FUNCTION_BLOCK EM_OutfeedModule EXTENDS CommonModule IMPLEMENTS I_OutfeedModule
VAR
	//Components
	Axis : FB_Component_BasicAxis;

	//
	_CmdOutfeed : ST_OutfeedCommand;
	_StsOutfeed : ST_OutfeedStatus;
	_CfgOutfeed : ST_OutfeedConfig;
	_RcpOutfeed : ST_OutfeedRecipe;

	//Test Vars
	Homed : BOOL;
END_VAR

PROPERTY CfgOutfeed : REFERENCE TO ST_OutfeedConfig
GET
CfgOutfeed REF= _CfgOutfeed;
END_GET
END_PROPERTY

PROPERTY CmdOutfeed : REFERENCE TO ST_OutfeedCommand
GET
CmdOutfeed REF= _CmdOutfeed;
END_GET
END_PROPERTY

METHOD PUBLIC CyclicLogic
IF NOT _InitComplete THEN
	_InitComplete := Initialize();
	RETURN;
END_IF

SUPER^.CyclicLogic();
END_METHOD

//! @summary This method contains code which will execute when this PackML module is in the <b>Execute</b> state
METHOD PROTECTED Execute
(*! <description> <b>The base implementation of this method is empty. User must override this method to provide functionality.</b>
<table> 
	<tr>
		<th> Previous State </th>
		<th> Transition In </th>
		<th> Transition Out </th>
		<th> Next State  </th> 
	</tr>
	<tr>
		<td> Starting<b>-or-</b>Unholding <b>-or-</b>Unsuspending</td>
		<td> State Complete<i>(Starting<b>-or-</b>Unholding<b>-or-</b>Unsuspending)</i></td> 
		<td> State Complete<b>-or-</b>Hold Command<b>-or-</b>Suspend Command</td>
		<td> Completing<b>-or-</b>Holding<b>-or-</b>Suspending</td>
	</tr>
</table>
This method is called as required by <c>StateControl()</c>
</description> 

*)
VAR
END_VAR
CASE _CurrentMode OF
	E_PMLCustomMode.Production:
		CASE DescendantSequenceState OF
			0:
				IF _StsOutfeed.ProductAtReady THEN
					DescendantSequenceState := DescendantSequenceState + 10;
				END_IF

			10:
				IF Axis.MoveVelocity(10.0, 0) THEN
					DescendantSequenceState := DescendantSequenceState + 10;
				END_IF

			20:
				IF Axis.Axis.Status.Moving THEN
					_StsOutfeed.ProductAtReady	:= FALSE;
					_StsOutfeed.ConveyorRunning := TRUE;
				END_IF

				IF _StsOutfeed.ProductRemoved THEN
					_CmdOutfeed.StopConveyor := FALSE;
					Axis.Stop();
					DescendantSequenceState := DescendantSequenceState + 10;
				END_IF

			30:
				IF Axis.Axis.Status.NotMoving THEN
					_StsOutfeed.ConveyorRunning := FALSE;
					DescendantSequenceState		:= 0;
				END_IF
		END_CASE

	E_PMLCustomMode.Home:
		CASE DescendantSequenceState OF
			0:
				IF _CmdCommon.Home AND NOT _StsCommon.Homed THEN
					_CmdCommon.Home := FALSE;
					Axis.Home();
					DescendantSequenceState := DescendantSequenceState + 10;
				END_IF

			10:
				IF Axis.Axis.Status.Homed THEN
					_StsCommon.Homed := TRUE;
				END_IF
		END_CASE
END_CASE

SUPER^.Execute();
END_METHOD

METHOD PROTECTED Initialize : BOOL
VAR
	i: UDINT;
END_VAR
Initialize := FALSE;
CASE DescendantSequenceState OF
	0: //Register Modules

		//Register Components
		RegisterComponent(Axis);

		//I_CommonModuleBase

		//I_CommonComponent
		ipComponents[1] := Axis;

		//Setup Config
		_LogModeChanges			:= FALSE;
		_LogStateChanges		:= FALSE;
		DescendantSequenceState := DescendantSequenceState + 10;

	10:
		// Copy Mode names
		FOR i := 1 TO 10 DO
			ModeNames[i] := F_UnitModeToString(UDINT_TO_DINT(i));
		END_FOR

		DescendantSequenceState := DescendantSequenceState + 10;

	20:
		//Initialize_Recipes();
		DescendantSequenceState := DescendantSequenceState + 10;

	30: // Call the Super 
		IF SUPER^.Initialize() THEN
			DescendantSequenceState := DescendantSequenceState + 10;
		END_IF

	40:
		Initialize := TRUE;
END_CASE
END_METHOD

PROPERTY RcpOutfeed : REFERENCE TO ST_OutfeedRecipe
GET
RcpOutfeed REF= _RcpOutfeed;
END_GET
END_PROPERTY

PROPERTY StsOutfeed : REFERENCE TO ST_OutfeedStatus
GET
StsOutfeed REF= _StsOutfeed;
END_GET
END_PROPERTY

END_FUNCTION_BLOCK

(* stored: Version 1.1.0.1, ProductVersion 3.1.4024.12
   POU EM_OutfeedModule: Id {7cfe66d8-35ba-4314-bc5b-79de6dfce221}, SpecialFunc None
   Folder I_CyclicLogic: Id {bff73ff0-91fb-43bc-8249-92d4b9647678}
   Folder I_OutfeedModule: Id {69613287-f892-473e-b1d8-0484c46e7d3a}
   Folder Initialize: Id {2f6fe5d0-4ad8-4db5-bcbb-919a2371bcc0}
   Folder Waiting: Id {90aacb5d-d031-4a9a-a8b9-804c40c70e47}
   Property CfgOutfeed: Id {a44dd973-0916-4949-a737-65d3485b91ec}
   Get Get: Id {319902ff-1362-472b-b229-c462e2493a5e}
   Property CmdOutfeed: Id {4c76f708-fd44-49ee-89dc-ce3046ef3f80}
   Get Get: Id {b3b04fb8-826d-4de2-b263-f0bc53875584}
   Method CyclicLogic: Id {4340cd9c-c928-4e0a-bb64-e13a6fc3c8ca}
   Method Execute: Id {72fd1940-d387-4987-ac34-491b6521b66b}
   Method Initialize: Id {5233c20d-7b9b-4059-b797-40c895a2027a}
   Property RcpOutfeed: Id {0b12ebb9-62cb-4cc2-b1ed-ede402f73212}
   Get Get: Id {b53521d8-ac70-4d27-bdae-fb2b00cfbf2b}
   Property StsOutfeed: Id {bf8eb5b2-3251-4d10-ad35-16de5a921b2c}
   Get Get: Id {b37dbd37-b31b-4a8d-9f29-40b363467d02} *)
